# EPICS autosave request: ipApp/Db/Leukos_laser_settings.req
$(P)$(R)Frequency
$(P)$(R)TriggerMode
$(P)$(R)ReadSettings.SCAN
